TYPE ST_CylinderX_Config :
    STRUCT
        ExtendTime  : LREAL;
        RetractTime : LREAL;
    END_STRUCT
END_TYPE

(* stored: Version 1.1.0.1
   DUT ST_CylinderX_Config: Id {960a85c6-bf60-4485-8329-866fbb31a19d} *)
